{attribute 'qualified_only'}
{attribute 'strict'}
TYPE DataSelector :
(
	_C 		:= 0,
	_V 		:= 1,
	_P		:= 2,
	_Q		:= 3,
	_S		:= 4,
	_E		:= 5,
	_F		:= 6	
);
END_TYPE

(* stored: Version 1.1.0.1, ProductVersion 3.1.4026.18
   DUT DataSelector: Id {63792fc6-4f5f-4584-bfe4-c68005034a28} *)
